{attribute 'qualified_only'}
{attribute 'strict'}
{attribute 'to_string'}
{info 'E_INSTANCE placeholder for process identification; add new members here'}
TYPE E_INSTANCE : // placeholder for process identification; add new members here
(
	INSTANCE_NULL,
  // list your process instances here
  INSTANCE_EXAMPLE,
  INSTANCE_MAX
)UINT;
END_TYPE

(* stored: Version 1.1.0.1, ProductVersion 3.1.4026.18
   DUT E_INSTANCE: Id {9bd75b71-2b5d-4f2b-b74f-2d020b4ae5e6} *)
